// TIA Portal V16 export
VAR_GLOBAL   // PLC tag table "Conveyor_IO_LAD"
   Conveyor_StartButton AT %I0.0 : Bool;
   Conveyor_StopOK AT %I0.1 : Bool;
   Conveyor_EStopOK AT %I0.2 : Bool;
   Conveyor_OverloadOK AT %I0.3 : Bool;
   Conveyor_JamSensor AT %I0.4 : Bool;
   Conveyor_ResetButton AT %I0.5 : Bool;
   Conveyor_MotorCmd AT %Q0.0 : Bool;
   Conveyor_RunLamp AT %Q0.1 : Bool;
   Conveyor_FaultLamp AT %Q0.2 : Bool;
END_VAR
